# EPICS substitutions: iocs/cpscIOC/iocBoot/ioccpscIOC/substitutions/canberra_13.substitutions
file "$(MCA)/mcaApp/Db/simple_mca.db"
{
pattern
{P           M       DTYP           INP         PREC  CHANS}
{cpscIOC:med:   mca1  "asynMCA"   "@asyn(AIM2/1 0)"    3  2048}
{cpscIOC:med:   mca2  "asynMCA"   "@asyn(AIM2/1 1)"    3  2048}
{cpscIOC:med:   mca3  "asynMCA"   "@asyn(AIM2/1 2)"    3  2048}
{cpscIOC:med:   mca4  "asynMCA"   "@asyn(AIM2/2 0)"    3  2048}
{cpscIOC:med:   mca5  "asynMCA"   "@asyn(AIM2/2 1)"    3  2048}
{cpscIOC:med:   mca6  "asynMCA"   "@asyn(AIM2/2 2)"    3  2048}
{cpscIOC:med:   mca7  "asynMCA"   "@asyn(AIM3/1 0)"    3  2048}
{cpscIOC:med:   mca8  "asynMCA"   "@asyn(AIM3/1 1)"    3  2048}
{cpscIOC:med:   mca9  "asynMCA"   "@asyn(AIM3/1 2)"    3  2048}
{cpscIOC:med:   mca10 "asynMCA"   "@asyn(AIM3/2 0)"    3  2048}
{cpscIOC:med:   mca11 "asynMCA"   "@asyn(AIM3/3 1)"    3  2048}
{cpscIOC:med:   mca12 "asynMCA"   "@asyn(AIM3/4 2)"    3  2048}
{cpscIOC:med:   mca13 "asynMCA"   "@asyn(AIM3/2 3)"    3  2048}
{cpscIOC:med:   mca0  "Soft Channel"   ""     3  2048}
}

file "$(MCA)/mcaApp/Db/icb_amp.db"
{
pattern
{P			AMP		PORT}
{cpscIOC:med:	amp1	"icbAmp1"}
{cpscIOC:med:	amp2	"icbAmp2"}
{cpscIOC:med:	amp3	"icbAmp3"}
{cpscIOC:med:	amp4	"icbAmp4"}
{cpscIOC:med:	amp5	"icbAmp5"}
{cpscIOC:med:	amp6	"icbAmp6"}
{cpscIOC:med:	amp7	"icbAmp7"}
{cpscIOC:med:	amp8	"icbAmp8"}
{cpscIOC:med:	amp9	"icbAmp9"}
{cpscIOC:med:	amp10	"icbAmp10"}
{cpscIOC:med:	amp11	"icbAmp11"}
{cpscIOC:med:	amp12	"icbAmp12"}
{cpscIOC:med:	amp13	"icbAmp13"}
}

file "$(MCA)/mcaApp/Db/icb_adc.db"
{
pattern
{P			ADC		PORT}
{cpscIOC:med:	adc1	"icbAdc1"}
{cpscIOC:med:	adc2	"icbAdc2"}
{cpscIOC:med:	adc3	"icbAdc3"}
{cpscIOC:med:	adc4	"icbAdc4"}
}

file "$(MCA)/mcaApp/Db/icb_hvps.db"
{
pattern
{P			HVPS	LIMIT	PORT}
{cpscIOC:med:	hvps1	1000	"icbHvps1"}
}
